(* Schneider Machine Expert - Basic project Exercise-5 - Multiple Switch with multiple Motors, file version 2.9.0.0 *)
(* ProjectInformations: Name=New project *)

HARDWARE
  Cpu 0: TM221M16R/G
  EthernetConfiguration: NetworkName=M221, IpAllocationMode=FixedAddress, IpAddress=0.0.0.0, SubnetMask=0.0.0.0
  SerialLineConfiguration: Baud=Baud19200, Parity=ParityEven, DataBits=DataBits8, StopBits=StopBits1, PhysicalMedium=PhysicalMediumRs485, TransmissionMode=TransmissionModeModbusRtu, SlaveId=1, Addressing=SlaveAddressing
  MastTask: UsePeriodScanMode=false, PeriodScan=100
  FastTask: Period=255
  CpuBehavior: StartingMode=StartAsPreviousState, AutoSaveRamOnEeprom=true, WatchdogPeriod=250

SYMBOLS  (address, symbol, comment, settings)
  %I0.0     SWITCH_1
  %I0.1     SWITCH_2
  %I0.2     SWITCH_3
  %I0.3     SWITCH_4
  %Q0.0     MOTOR_1
  %Q0.1     MOTOR_2
  %Q0.2     MOTOR_3
  %Q0.3     MOTOR_4

POU New POU
  (* SectionNumber=1 *)

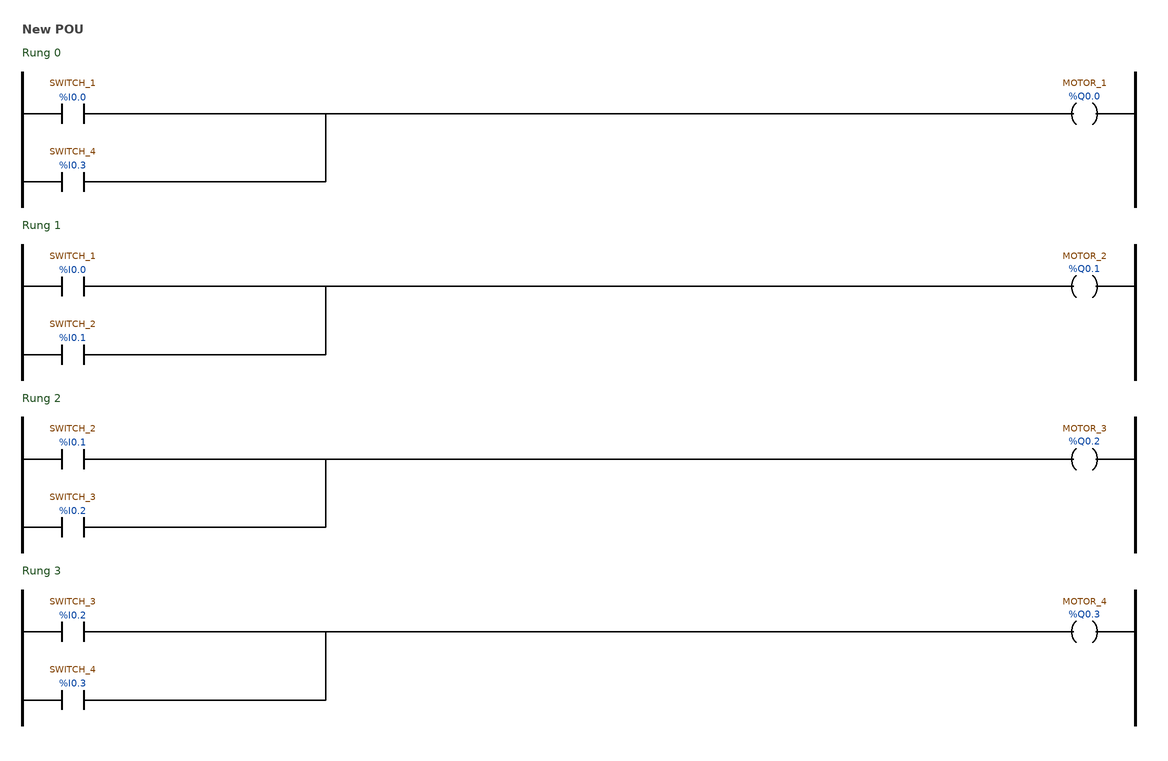

// Rung 0
  LD %I0.0                (* SWITCH_1 *)
  OR %I0.3                (* SWITCH_4 *)
  ST %Q0.0                (* MOTOR_1 *)
  // as ST:
  //   MOTOR_1 := SWITCH_1 OR SWITCH_4;

// Rung 1
  LD %I0.0                (* SWITCH_1 *)
  OR %I0.1                (* SWITCH_2 *)
  ST %Q0.1                (* MOTOR_2 *)
  // as ST:
  //   MOTOR_2 := SWITCH_1 OR SWITCH_2;

// Rung 2
  LD %I0.1                (* SWITCH_2 *)
  OR %I0.2                (* SWITCH_3 *)
  ST %Q0.2                (* MOTOR_3 *)
  // as ST:
  //   MOTOR_3 := SWITCH_2 OR SWITCH_3;

// Rung 3
  LD %I0.2                (* SWITCH_3 *)
  OR %I0.3                (* SWITCH_4 *)
  ST %Q0.3                (* MOTOR_4 *)
  // as ST:
  //   MOTOR_4 := SWITCH_3 OR SWITCH_4;
